# EPICS IOC start-up script: iocBoot/iocoh26/iocsh/wrist_cam.iocsh
#- INSTANCE  - Used for Camera Port Name and detector pv name
#- XSIZE     - Image Width
#- YSIZE     - Image Height
#- TYPE      - Image Datatype, default: Int8
#- COLORS    - Number of colors, default: 1

epicsEnvSet("EPICS_DB_INCLUDE_PATH", "$(EPICS_DB_INCLUDE_PATH):$(ADCORE)/db:$(ADURL)/db")

# Create a URL driver
# URLDriverConfig(const char *portName, int maxBuffers, size_t maxMemory,
#                 int priority, int stackSize)
URLDriverConfig("$(INSTANCE)", 0, 0)
dbLoadRecords("$(ADURL)/db/URLDriver.template","P=$(PREFIX),R=$(INSTANCE):,PORT=$(INSTANCE),ADDR=0,TIMEOUT=1")

# Create a standard arrays plugin.
NDStdArraysConfigure("Image1", 3, 0, "$(INSTANCE)", 0)

#Create a standard arrays plugin, set it to get data from first simDetector driver.
NDStdArraysConfigure("$(INSTANCE)Image", 3, 0, "$(INSTANCE)", 0, 2000000)

# Need to determine certain values from input parameters
iocshRun('epicsEnvSet("__FTVL", "$($(TYPE=Int8)_VAL)")', "Int8_VAL=UCHAR, UInt8_VAL=UCHAR, Int16_VAL=SHORT, UInt16_VAL=SHORT, Int32_VAL=LONG, UInt32_VAL=LONG, Float32_VAL=DOUBLE, Float64_VAL=DOUBLE")
iocshRun('epicsEnvSet("__TYPE", "$($(TYPE=Int8)_VAL)")', "Int8_VAL=Int8, UInt8_VAL=Int8, Int16_VAL=Int16, UInt16_VAL=Int16, Int32_VAL=Int32, UInt32_VAL=Int32, Float32_VAL=Float32, Float64_VAL=Float64")
luaCmd("epicsEnvSet('__SIZE', tostring((COLORS*XSIZE*YSIZE)|0))", "COLORS=$(COLORS=1), XSIZE=$(XSIZE), YSIZE=$(YSIZE)")

dbLoadRecords("$(ADCORE)/ADApp/Db/NDStdArrays.template", "P=$(PREFIX),R=image1:,PORT=$(INSTANCE)Image,ADDR=0,TIMEOUT=1,NDARRAY_PORT=$(INSTANCE),TYPE=$(__TYPE),FTVL=$(__FTVL),NELEMENTS=$(__SIZE)")

epicsEnvUnset("__FTVL")
epicsEnvUnset("__TYPE")
epicsEnvUnset("__SIZE")

# Load some AD plugins

# Don't need everything in here
# iocshLoad("$(ADCORE)/iocBoot/commonPlugins.cmd", "PREFIX=$(PREFIX), PORT=$(INSTANCE), QSIZE=20, XSIZE=$(XSIZE), YSIZE=$(YSIZE), NCHANS=1024, CBUFFS=20, MAX_THREADS=5")

# Create a JPEG file saving plugin
NDFileJPEGConfigure("FileJPEG1", $(QSIZE=20), 0, "$(INSTANCE)", 0)
dbLoadRecords("NDFileJPEG.template",  "P=$(PREFIX),R=JPEG1:,PORT=FileJPEG1,ADDR=0,TIMEOUT=1,NDARRAY_PORT=$(INSTANCE)")

# Load NDPluginPva plugin
NDPvaConfigure("PVA1", $(QSIZE=20), 0, "$(INSTANCE)", 0, $(PREFIX)Pva1:Image, 0, 0, 0)
dbLoadRecords("NDPva.template",  "P=$(PREFIX),R=Pva1:, PORT=PVA1,ADDR=0,TIMEOUT=1,NDARRAY_PORT=$(INSTANCE)")
#Must start PVA server if this is enabled
startPVAServer

# autosave stuff
# done already in common.iocsh?
# set_requestfile_path("./")
# set_requestfile_path("$(ADCORE)/db")
# set_requestfile_path("$(ADCORE)/iocBoot")
# set_requestfile_path("$(AUTOSAVE)/db")
# set_savefile_path("./autosave")
# set_pass0_restoreFile("auto_settings.sav")
# set_pass1_restoreFile("auto_settings.sav")
# save_restoreSet_status_prefix("$(PREFIX)")
# dbLoadRecords("$(AUTOSAVE)/db/save_restoreStatus.db", "P=$(PREFIX)")
# dbLoadRecords("$(AUTOSAVE)/db/configMenu.db", "P=$(PREFIX), CONFIG=ADAutoSave")
# set_requestfile_path("$(ADURL)/db")

# # Optional: load scan records
# dbLoadRecords("$(SSCAN)/db/scan.db", "P=$(PREFIX),MAXPTS1=2000,MAXPTS2=200,MAXPTS3=20,MAXPTS4=10,MAXPTSH=10")
# set_requestfile_path("$(SSCAN)/db")

# # Optional: load sseq record for acquisition sequence
# dbLoadRecords("$(CALC)/db/sseqRecord.db", "P=$(PREFIX), S=AcquireSequence")
# set_requestfile_path("$(CALC)/db")

# # Optional: load devIocStats records (requires DEVIOCSTATS module)
# dbLoadRecords("$(DEVIOCSTATS)/db/iocAdminSoft.db", "IOC=$(PREFIX)")

# # Optional: load alive record (requires ALIVE module)
# dbLoadRecords("$(ALIVE)/db/alive.db", "P=$(PREFIX),RHOST=164.54.100.11")

# Set the callback queue size to 5000, up from default of 2000 in base.
# This can be needed to avoid errors "callbackRequest: cbLow ring buffer full".
callbackSetQueueSize(5000)
